// TIA Portal V19 export
TYPE "LEXCHANGETRAY_typePc_Interface"
// stored: Access Published
   STRUCT
      sim { S7_SetPoint := 'True'} : "LEXCHANGETRAY_typePc_sim";   // simulate
      monitor { S7_SetPoint := 'True'} : "LEXCHANGETRAY_typePc_Monitor";   // 托盘状态
   END_STRUCT;
END_TYPE
